{attribute 'OPC.UA.DA' := '1'}    
TYPE ST_DO :
STRUCT
		Value		  AT %Q*	: BOOL	;
		Description 			: STRING	;

END_STRUCT
END_TYPE

(* stored: Version 1.1.0.1, ProductVersion 3.1.4024.12
   DUT ST_DO: Id {552d99e6-cdd3-4003-ac15-aaeab6e4cbf4} *)
